FUNCTION_BLOCK trip_controller_no_timer (* Composite Function Block Type *)
  (* Standard: 61499-2 *)
  (* Version 0.0, 11/29/2016, gulzha, nxtControl GmbH, template *)
  PACKAGE Main;
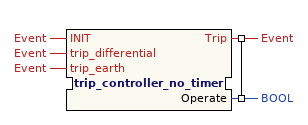
  EVENT_INPUT
    INIT; (* Initialization Request *)
    trip_differential; (* Normal Execution Request *)
    trip_earth; (* Normal Execution Request *)
  END_EVENT
  EVENT_OUTPUT
    Trip WITH Operate; (* Execution Confirmation *)
  END_EVENT
  VAR_OUTPUT
    Operate : BOOL; (* Current Output State *)
  END_VAR
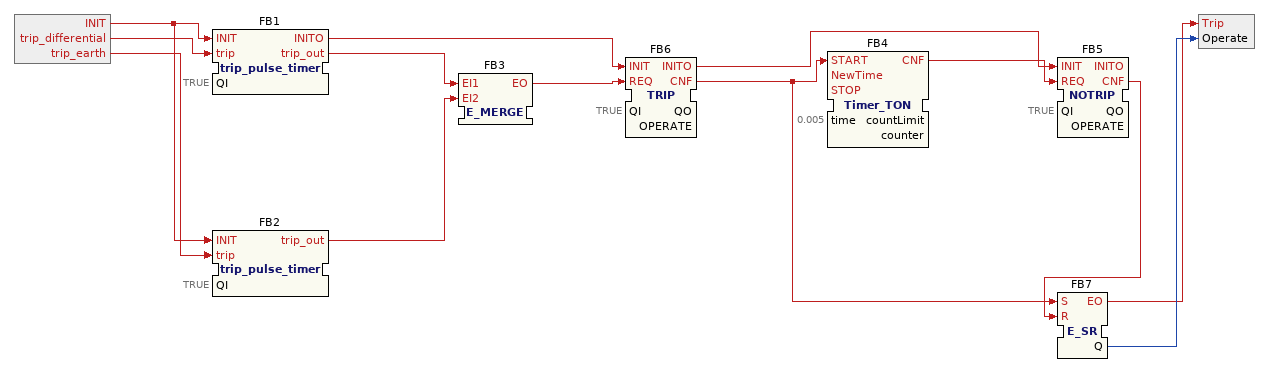
  FBS
    FB1 : trip_pulse_timer(QI := TRUE);
    FB2 : trip_pulse_timer(QI := TRUE);
    FB4 : Timer_TON(time := 0.005);
    FB5 : NOTRIP(QI := TRUE);
    FB6 : TRIP(QI := TRUE);
    FB7 : E_SR;
    FB3 : E_MERGE;
  END_FBS
  EVENT_CONNECTIONS
    FB4.CNF TO FB5.REQ;
    FB6.CNF TO FB4.START;
    FB6.CNF TO FB7.S;
    FB5.CNF TO FB7.R;
    FB7.EO TO Trip;
    FB1.INITO TO FB6.INIT;
    FB6.INITO TO FB5.INIT;
    FB1.trip_out TO FB3.EI1;
    FB2.trip_out TO FB3.EI2;
    FB3.EO TO FB6.REQ;
    INIT TO FB1.INIT;
    INIT TO FB2.INIT;
    trip_differential TO FB1.trip;
    trip_earth TO FB2.trip;
  END_CONNECTIONS
  DATA_CONNECTIONS
    FB7.Q TO Operate;
  END_CONNECTIONS
END_FUNCTION_BLOCK
